// Mitsubishi GX Works2 project: s   PLC: FX3U/FX3UC

PROGRAM MAIN
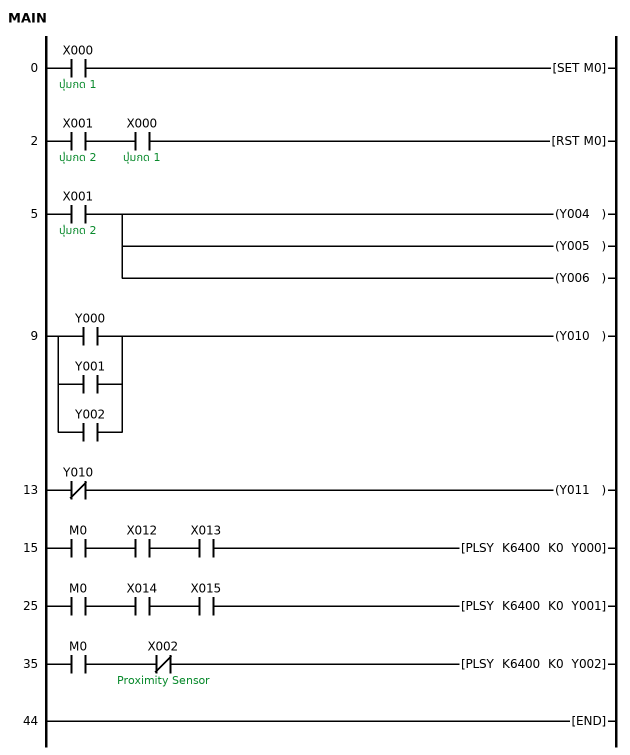
0     LD      X000  ; ปุ่มกด 1
      SET     M0
2     LD      X001  ; ปุ่มกด 2
      AND     X000  ; ปุ่มกด 1
      RST     M0
5     LD      X001  ; ปุ่มกด 2
      OUT     Y004
      OUT     Y005
      OUT     Y006
9     LD      Y000
      OR      Y001
      OR      Y002
      OUT     Y010
13    LDI     Y010
      OUT     Y011
15    LD      M0
      AND     X012
      AND     X013
      PLSY    K6400 K0 Y000
25    LD      M0
      AND     X014
      AND     X015
      PLSY    K6400 K0 Y001
35    LD      M0
      ANI     X002  ; Proximity Sensor
      PLSY    K6400 K0 Y002
44    END
END_PROGRAM
